# EPICS autosave request: ipApp/Db/JenaNV100D_settings.req
# Jena NV100/D
$(P)$(C)write
$(P)$(C)write.PREC
$(P)$(C)read.DESC
$(P)$(C)read.PREC
$(P)$(C)read.SCAN
$(P)$(C)cl
$(P)$(C)kp
$(P)$(C)kp_RBV.SCAN
$(P)$(C)ki
$(P)$(C)ki_RBV.SCAN
$(P)$(C)kd
$(P)$(C)kd_RBV.SCAN
